// TIA Portal V17 export
// export: Created 2025-03-05T08:01:12.1315007Z, ExportSetting WithDefaults, DisplayName Totally Integrated Automation Portal, DisplayVersion V17 Update 8, DisplayName TIA Portal Openness, DisplayVersion V17 Update 8, DisplayName TIA Portal Version Control Interface, DisplayVersion V17, DisplayName SINAMICS Startdrive Advanced, DisplayVersion V17 SP2, DisplayName SINAMICS Startdrive G110M, G120, G120C, G120D, G120P, G115D, DisplayVersion V17 SP2, DisplayName SINAMICS Startdrive G130, G150, S120, S150, SINAMICS MV, S210, DisplayVersion V17 SP2, DisplayName STEP 7 Professional, DisplayVersion V17 Update 8, DisplayName SINUMERIK ONE STEP 7 Toolbox, DisplayVersion V17 Update 12, DisplayName SINUMERIK 840D sl STEP 7 Toolbox, DisplayVersion V17 Update 12, DisplayName STEP 7 Safety, DisplayVersion V17 Update 6, DisplayName WinCC Advanced, DisplayVersion V17 Update 8
FUNCTION "FC2200_NETWORKS" : Void   // FC2200, LAD
TITLE = NETWORK BLOCKS
{ S7_Optimized_Access := 'FALSE' }
AUTHOR : ETXETAR
VERSION : 1.0
// stored: AutoNumber false, IsIECCheckEnabled false, SetENOAutomatically false, UDAEnableTagReadback false
BEGIN

REGION Network 1: CALL FC2202 PROFINET
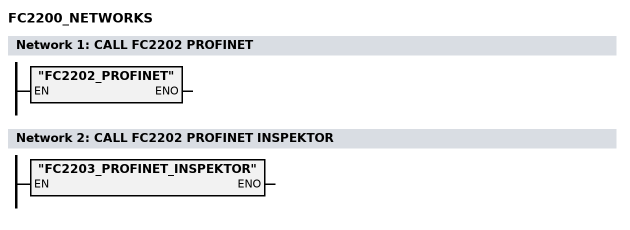
   RUNG wire#powerrail
      "FC2202_PROFINET"()
   END_RUNG
   // the same network as SCL:
   "FC2202_PROFINET"();
END_REGION

REGION Network 2: CALL FC2202 PROFINET INSPEKTOR
   RUNG wire#powerrail
      "FC2203_PROFINET_INSPEKTOR"()
   END_RUNG
   // the same network as SCL:
   "FC2203_PROFINET_INSPEKTOR"();
END_REGION
END_FUNCTION
